{attribute 'qualified_only'}
VAR_GLOBAL
	fbSoftWash : FB_SoftWash;
	fbNormalWash : FB_NormalWash;
	fbHeavyWash : FB_HeavyWash;
	
	fbMotor : FB_BaseMotor;
	fbWaterController : FB_WaterController;
END_VAR

(* stored: Version 1.1.0.1, ProductVersion 3.1.4024.16
   GVL GVL_References: Id {b44de6da-9732-49ef-9607-d87e175c08b8} *)
